FUNCTION_BLOCK FB_AutomaticControlWinch
VAR_INPUT
	bEnable 							: BOOL;
	bStartMotion 						: BOOL;
	bStopMotion 						: BOOL;
	stMotionReferenceGeneratorSettings  : ST_MotionReferenceGeneratorSettings;
	stAutomaticControlSettings 			: ST_AutomaticControlSettings;
	stClosedLoopControlSettings 		: ST_ClosedLoopControlSettings;
	stOpenLoopControlSettings			: ST_OpenLoopControlSettings;
	stParam 							: ST_Parameters; 
	fPositionFeedback					: LREAL;
END_VAR
VAR_OUTPUT
	fTime : LREAL;
	fVelocityReference_ms : LREAL;
	fPositionReference_m : LREAL;
	fControlOutputNormalized : LREAL;
	fPositionError_mm : LREAL;
END_VAR
VAR
	fbClock : FB_Clock;	
	fbMotionReferenceGenerator 		: FB_MotionReferenceGenerator_limit;	
	fbVelocityFeedForwardControl 	: FB_OpenLoopControlWinch;
	fbResetIntegralController 		: FB_ResetIntegralController; 
	fbClosedLoopPositionControl 	: FB_ClosedLoopControl;
END_VAR

fbClock(
	bEnable := bEnable,
	bStart := bStartMotion,
	bStop := bStopMotion,
	fCycleTime := G_Parameters.stParam.fCyclicTime
);

fbMotionReferenceGenerator(
	bEnable := bEnable,
	stMotionReferenceGeneratorSettings := stMotionReferenceGeneratorSettings,
	fClock_s := fbClock.fTime
);

fbVelocityFeedForwardControl(
	bEnable := stAutomaticControlSettings.bEnableVelocityFeedForwardControl,
	fInput_ms := fbMotionReferenceGenerator.fVelocityReference_ms,
	fDisplacment_cc := stParam.fDisplacment_cc,
	fLin_m_ToRot_deg_Scaling := stParam.fWinchDrumScaling,
	stOpenLoopControlSettings := stOpenLoopControlSettings
);

fbResetIntegralController(
	stClosedLoopControlSettings := stClosedLoopControlSettings,
	fPositionError_m := fbClosedLoopPositionControl.fPositionError,
	fVelocityReference_ms := fbMotionReferenceGenerator.fVelocityReference_ms
);

fbClosedLoopPositionControl(
	bEnable := stAutomaticControlSettings.bEnableClosedLoopPositionControl,
	stParam := stParam,
	stClosedLoopControlSettings := stClosedLoopControlSettings,		
	bActivateIntegralController := stAutomaticControlSettings.bEnableIntegralController,
	bIntegralControllReset := fbResetIntegralController.bReset,
	fInput_m := fbMotionReferenceGenerator.fPositionReference_m,
	fFeedback_m := fPositionFeedback
);

fVelocityReference_ms := fbMotionReferenceGenerator.fVelocityReference_ms;
fPositionReference_m := fbMotionReferenceGenerator.fPositionReference_m;
fTime := fbClock.fTime;
fPositionError_mm := fbClosedLoopPositionControl.fPositionError*1E3;

IF bEnable THEN
	fControlOutputNormalized := LIMIT(-1.0, (fbVelocityFeedForwardControl.fNormalizedOutput + fbClosedLoopPositionControl.fNormalizedOutput), 1.0);
ELSE
	fControlOutputNormalized := 0.0;
END_IF

END_FUNCTION_BLOCK

(* stored: Version 1.1.0.1, ProductVersion 3.1.4024.11
   POU FB_AutomaticControlWinch: Id {fd6f8a87-c5d5-4f70-8249-2b0de500d6fe}, SpecialFunc None *)
